# EPICS substitutions: rbd9103App/Db/rbd9103.substitutions
file "$(ASYN)/db/asynRecord.db"
{
pattern { P,       R,          PORT,    ADDR, OMAX, IMAX }
        { "DEV:", "RBD9103:AsynIO", "RBD_TTY", "0", "0", "0" }
}

file "$(RBD_9103)/db/rbd9103.template"
{
pattern { P,     R,          PORT}
        {"DEV:", "RBD9103:", "RBD"}
}

file "$(RBD_9103)/db/rbd9103_recording.template"
{
pattern { P,     R,          PORT}
        {"DEV:", "RBD9103:", "RBD"}
}
